PROGRAM DRIVE_Controller
VAR
	eJogMode: 				E_JogMode;
	fbAxisControls:			ARRAY [1..CE_AXIS_C] OF FB_AxisControl;
	
END_VAR

IF (G_xManualMoveMode) THEN
	eJogMode:= MC_JOGMODE_CONTINOUS;
ELSE
	eJogMode:= MC_JOGMODE_INCHING;
END_IF

X_Drive_ACT();
Y_Drive_ACT();
Z_Drive_ACT();
C_Drive_ACT();

ACTION C_Drive_ACT:
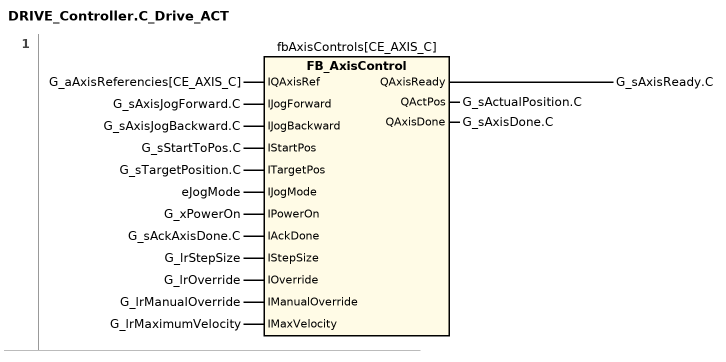
// NETWORK 1
fbAxisControls[CE_AXIS_C](
    IQAxisRef := G_aAxisReferencies[CE_AXIS_C],
    IJogForward := G_sAxisJogForward.C,
    IJogBackward := G_sAxisJogBackward.C,
    IStartPos := G_sStartToPos.C,
    ITargetPos := G_sTargetPosition.C,
    IJogMode := eJogMode,
    IPowerOn := G_xPowerOn,
    IAckDone := G_sAckAxisDone.C,
    IStepSize := G_lrStepSize,
    IOverride := G_lrOverride,
    IManualOverride := G_lrManualOverride,
    IMaxVelocity := G_lrMaximumVelocity,
    QActPos => G_sActualPosition.C,
    QAxisDone => G_sAxisDone.C); // FB_AxisControl
G_sAxisReady.C := fbAxisControls[CE_AXIS_C].QAxisReady;
END_ACTION

ACTION X_Drive_ACT:
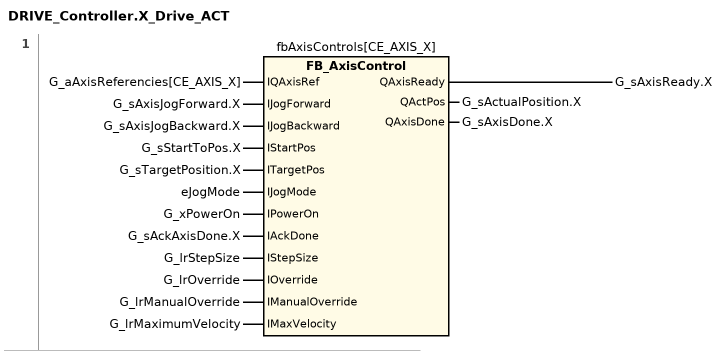
// NETWORK 1
fbAxisControls[CE_AXIS_X](
    IQAxisRef := G_aAxisReferencies[CE_AXIS_X],
    IJogForward := G_sAxisJogForward.X,
    IJogBackward := G_sAxisJogBackward.X,
    IStartPos := G_sStartToPos.X,
    ITargetPos := G_sTargetPosition.X,
    IJogMode := eJogMode,
    IPowerOn := G_xPowerOn,
    IAckDone := G_sAckAxisDone.X,
    IStepSize := G_lrStepSize,
    IOverride := G_lrOverride,
    IManualOverride := G_lrManualOverride,
    IMaxVelocity := G_lrMaximumVelocity,
    QActPos => G_sActualPosition.X,
    QAxisDone => G_sAxisDone.X); // FB_AxisControl
G_sAxisReady.X := fbAxisControls[CE_AXIS_X].QAxisReady;
END_ACTION

ACTION Y_Drive_ACT:
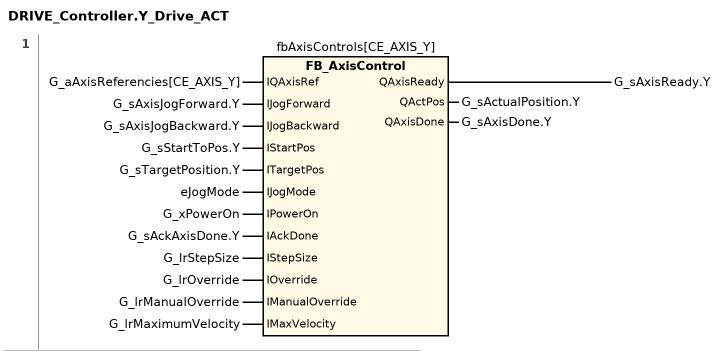
// NETWORK 1
fbAxisControls[CE_AXIS_Y](
    IQAxisRef := G_aAxisReferencies[CE_AXIS_Y],
    IJogForward := G_sAxisJogForward.Y,
    IJogBackward := G_sAxisJogBackward.Y,
    IStartPos := G_sStartToPos.Y,
    ITargetPos := G_sTargetPosition.Y,
    IJogMode := eJogMode,
    IPowerOn := G_xPowerOn,
    IAckDone := G_sAckAxisDone.Y,
    IStepSize := G_lrStepSize,
    IOverride := G_lrOverride,
    IManualOverride := G_lrManualOverride,
    IMaxVelocity := G_lrMaximumVelocity,
    QActPos => G_sActualPosition.Y,
    QAxisDone => G_sAxisDone.Y); // FB_AxisControl
G_sAxisReady.Y := fbAxisControls[CE_AXIS_Y].QAxisReady;
END_ACTION

ACTION Z_Drive_ACT:
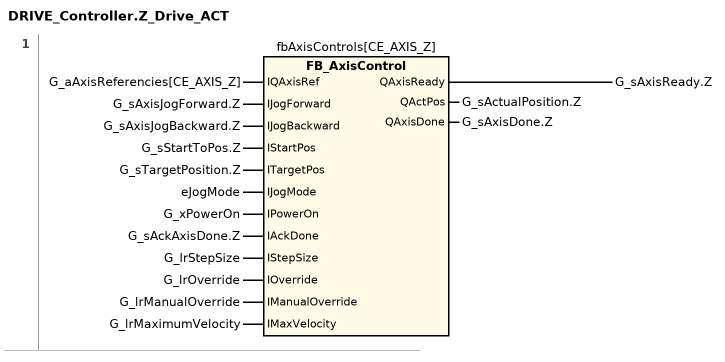
// NETWORK 1
fbAxisControls[CE_AXIS_Z](
    IQAxisRef := G_aAxisReferencies[CE_AXIS_Z],
    IJogForward := G_sAxisJogForward.Z,
    IJogBackward := G_sAxisJogBackward.Z,
    IStartPos := G_sStartToPos.Z,
    ITargetPos := G_sTargetPosition.Z,
    IJogMode := eJogMode,
    IPowerOn := G_xPowerOn,
    IAckDone := G_sAckAxisDone.Z,
    IStepSize := G_lrStepSize,
    IOverride := G_lrOverride,
    IManualOverride := G_lrManualOverride,
    IMaxVelocity := G_lrMaximumVelocity,
    QActPos => G_sActualPosition.Z,
    QAxisDone => G_sAxisDone.Z); // FB_AxisControl
G_sAxisReady.Z := fbAxisControls[CE_AXIS_Z].QAxisReady;
END_ACTION

END_PROGRAM

(* stored: Version 1.1.0.1, ProductVersion 3.1.4022.18
   POU DRIVE_Controller: Id {0b4b4fbb-55f4-4fa6-9595-368ee27aa716}, SpecialFunc None
   Action C_Drive_ACT: Id {1f644ece-d39b-4854-ab3e-b53e96db81a3}
   Action X_Drive_ACT: Id {fb1c16d4-804e-4173-935b-da2b262fc4d0}
   Action Y_Drive_ACT: Id {65d26bee-92d5-4bda-92db-d57007d02104}
   Action Z_Drive_ACT: Id {802af4c2-4bcb-4e28-a358-7f30f2913201} *)
